{attribute 'linkalways'} 
{attribute 'no_explicit_call' := 'This FB is a CLASS and must be accessed using methods or properties'}
{attribute 'enable_dynamic_creation'}
FUNCTION_BLOCK Node_F_VN_FillContainerExp_ITcVnImage EXTENDS VisionNode
VAR
    ipContainer : _ITcVnContainer;
    ipValue : _ITcVnImage;
    nStartIdx : _ULINT(0);
    nCount : _ULINT(0);
    hrPrev : _HRESULT(S_OK);
    hresult : _HRESULT(S_OK);
END_VAR

METHOD PUBLIC  Clone : I_Node
VAR
    pNode : POINTER TO Node_F_VN_FillContainerExp_ITcVnImage;
END_VAR
pNode := __NEW(Node_F_VN_FillContainerExp_ITcVnImage);
Clone := pNode^;
END_METHOD

METHOD FB_init : BOOL
VAR_INPUT
    bInitRetains : BOOL; // if TRUE, the retain variables are initialized (warm start / cold start)
    bInCopyCode : BOOL;  // if TRUE, the instance afterwards gets moved into the copy code (online change)
END_VAR
AddInput('ipContainer', ipContainer);
AddInput('ipValue', ipValue);
AddParameter('nStartIdx', nStartIdx);
AddParameter('nCount', nCount);
AddInput('hrPrev', hrPrev);
AddOutput('ipContainer', ipContainer);
AddOutput('hresult',hresult);
END_METHOD

METHOD PROTECTED OnExecute
hresult.Value := F_VN_FillContainerExp_ITcVnImage(
    ipContainer := ipContainer.Value,
    ipValue := ipValue.Value,
    nStartIdx := nStartIdx.Value,
    nCount := nCount.Value,
    hrPrev:= hrPrev.Value);
END_METHOD

METHOD PUBLIC PreExecutionCheck
VAR_INPUT
    Check : I_PreExecutionChecks;
END_VAR
Check.IsTrue(ipContainer.IsValid, 'ipContainer must be a valid container');
Check.IsTrue(ipContainer.IsType(TC_GLOBAL_CONST_LIST.ContainerType_Vector_ITcVnImage), 'ipContainer contains incorrect type');
END_METHOD

END_FUNCTION_BLOCK

(* stored: Version 1.1.0.1, ProductVersion 3.1.4026.13
   POU Node_F_VN_FillContainerExp_ITcVnImage: Id {f9f73891-97ef-4403-a0e9-5dd75a8c049d}, SpecialFunc None
   Folder Constructor: Id {b416f94f-0354-4361-80d2-3e75abe58dd9}
   Method Clone: Id {c3908b35-2949-429d-9ddb-78ef7dad8022}
   Method FB_init: Id {be549b95-de7a-496a-8994-d1543dbbe3c6}
   Method OnExecute: Id {5b173151-a59f-40d2-9f3f-02665f325737}
   Method PreExecutionCheck: Id {4e52ba38-7972-4d8a-b71d-5f9168392a35} *)
